// TIA Portal project "Serial_FB" (V15)

(* hardware
DEVICE "S7-1200 station_1"  S7-1200 Station
   slot 0: "Rack_0"  S7-1200 Rack  Rack  V1.0
   slot 1: "PLC_1"  CPU 1215C DC/DC/DC  6ES7 215-1AG40-0XB0  V4.2
DEVICE "HMI_1"  TP1200 Comfort
   slot 0: "HMI_1"  TP1200 Comfort  6AV2 124-0MC01-0AX0  15.0.0.0
   slot 1: "HMI_RT_1"  TP1200 Comfort  6AV2 124-0MC01-0AX0  15.0.0.0
   slot 5: "HMI_1.IE_CP_1"  PROFINET Interface  15.0.0.0
      slot 1: "PROFINET Interface_1"  PROFINET Interface
         slot 1: "Port_1"  Port
         slot 2: "Port_2"  Port
   slot 7: "HMI_1.MPI/DP_CP_1"  MPI/DP Interface  15.0.0.0
*)

// ===== PLC "PLC_1"  CPU 1215C DC/DC/DC =====

VAR_GLOBAL   // PLC tag table "Default tag table"
   "Begin_M" AT %M0.0 : Bool;
   "Pin_Out" AT %Q0.0 : Bool;
   "Port_Out" AT %QB0 : SInt;
   "Transfer_Status" AT %M0.1 : Bool;
   "Receive_Status" AT %M0.2 : Bool;
   "Start_M" AT %M0.3 : Bool;
   "Received_Byte" AT %MB2 : Byte;
END_VAR

DATA_BLOCK "Transmit_DB"   // DB2
{ S7_Optimized_Access := 'TRUE' }
VERSION : 0.1
// stored: InstanceOfName Transmit
"Transmit"
BEGIN
END_DATA_BLOCK

DATA_BLOCK "Receive_DB"   // DB4
{ S7_Optimized_Access := 'TRUE' }
VERSION : 0.1
// stored: InstanceOfName Receive
"Receive"
BEGIN
END_DATA_BLOCK

DATA_BLOCK "Input_48_Bit"   // DB5
{ S7_Optimized_Access := 'TRUE' }
VERSION : 0.1
   VAR RETAIN
      DI : Array[0..47] of Bool;
   END_VAR
BEGIN
END_DATA_BLOCK

// folder: System blocks/Program resources

DATA_BLOCK "Timer_1"   // DB1
{ S7_Optimized_Access := 'TRUE' }
AUTHOR : Simatic
FAMILY : IEC
NAME : IEC_TMR
VERSION : 1.0
// stored: InstanceOfName IEC_TIMER
"IEC_TIMER"
BEGIN
END_DATA_BLOCK

DATA_BLOCK "Timer_2"   // DB3
{ S7_Optimized_Access := 'TRUE' }
AUTHOR : Simatic
FAMILY : IEC
NAME : IEC_TMR
VERSION : 1.0
// stored: InstanceOfName IEC_TIMER
"IEC_TIMER"
BEGIN
END_DATA_BLOCK

// folder: (top level)

FUNCTION_BLOCK "Transmit"   // FB1, LAD
TITLE = Transmit 1 byte data serially to an output pin
{ S7_Optimized_Access := 'TRUE' }
VERSION : 0.1
   VAR_INPUT
      Data_In : Byte;
      "Begin" : Bool;
   END_VAR
   VAR_OUTPUT
      Serial_Out : Bool;
      Status : Bool;   // 1=In Progress, 0=Idle
   END_VAR
   VAR RETAIN
      Buffer : Array[0..9] of Bool;
      Temp : Byte;
      Clock : Time;
      i : DInt;
   END_VAR
   VAR_TEMP   // added for the SCL form of the ladder/FBD networks
      _w1 : Bool;
   END_VAR
   // Buffer[0] := true;
BEGIN

REGION Network 1: 1st bit of the input data
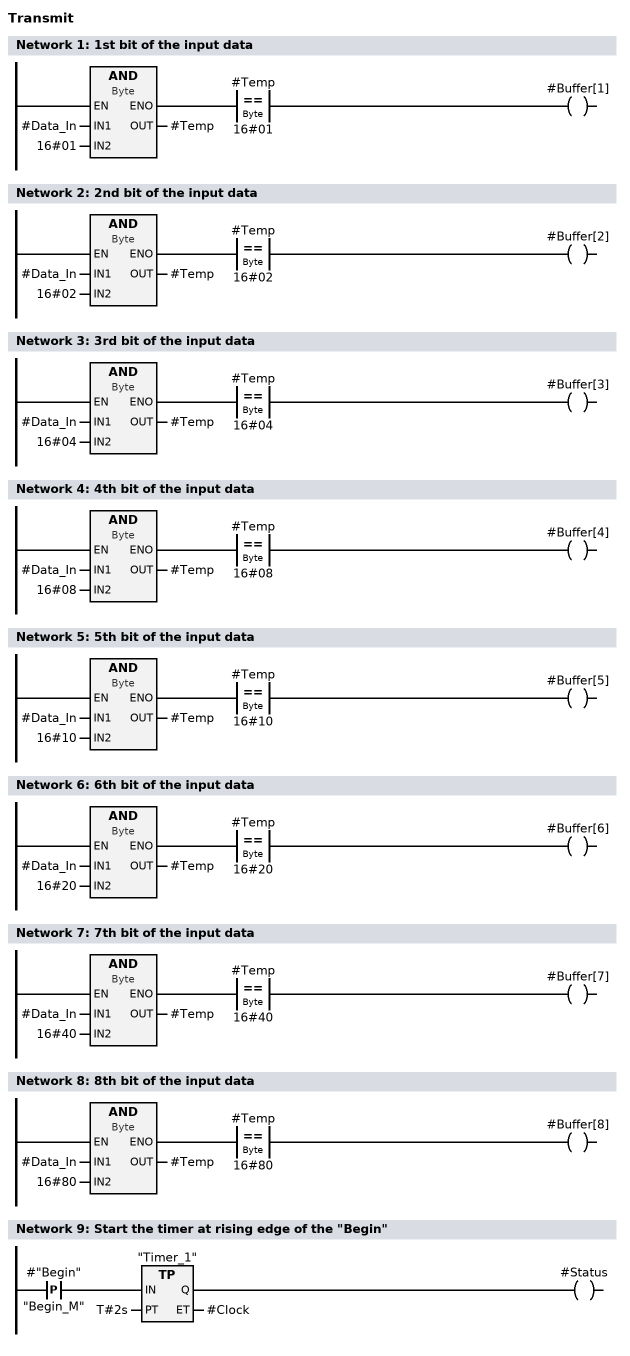
   RUNG wire#powerrail
      { S7_Templates := "SrcType := Byte" } And(in1 := #Data_In, in2 := 16#01, out => #Temp)
      { S7_Templates := "SrcType := Byte" } EQ_Contact(in1 := #Temp, in2 := 16#01)
      Coil( #Buffer[1] )
   END_RUNG
   // the same network as SCL:
   #Temp := #Data_In AND 16#01;
   #Buffer[1] := #Temp = 16#01;
END_REGION

REGION Network 2: 2nd bit of the input data
   RUNG wire#powerrail
      { S7_Templates := "SrcType := Byte" } And(in1 := #Data_In, in2 := 16#02, out => #Temp)
      { S7_Templates := "SrcType := Byte" } EQ_Contact(in1 := #Temp, in2 := 16#02)
      Coil( #Buffer[2] )
   END_RUNG
   // the same network as SCL:
   #Temp := #Data_In AND 16#02;
   #Buffer[2] := #Temp = 16#02;
END_REGION

REGION Network 3: 3rd bit of the input data
   RUNG wire#powerrail
      { S7_Templates := "SrcType := Byte" } And(in1 := #Data_In, in2 := 16#04, out => #Temp)
      { S7_Templates := "SrcType := Byte" } EQ_Contact(in1 := #Temp, in2 := 16#04)
      Coil( #Buffer[3] )
   END_RUNG
   // the same network as SCL:
   #Temp := #Data_In AND 16#04;
   #Buffer[3] := #Temp = 16#04;
END_REGION

REGION Network 4: 4th bit of the input data
   RUNG wire#powerrail
      { S7_Templates := "SrcType := Byte" } And(in1 := #Data_In, in2 := 16#08, out => #Temp)
      { S7_Templates := "SrcType := Byte" } EQ_Contact(in1 := #Temp, in2 := 16#08)
      Coil( #Buffer[4] )
   END_RUNG
   // the same network as SCL:
   #Temp := #Data_In AND 16#08;
   #Buffer[4] := #Temp = 16#08;
END_REGION

REGION Network 5: 5th bit of the input data
   RUNG wire#powerrail
      { S7_Templates := "SrcType := Byte" } And(in1 := #Data_In, in2 := 16#10, out => #Temp)
      { S7_Templates := "SrcType := Byte" } EQ_Contact(in1 := #Temp, in2 := 16#10)
      Coil( #Buffer[5] )
   END_RUNG
   // the same network as SCL:
   #Temp := #Data_In AND 16#10;
   #Buffer[5] := #Temp = 16#10;
END_REGION

REGION Network 6: 6th bit of the input data
   RUNG wire#powerrail
      { S7_Templates := "SrcType := Byte" } And(in1 := #Data_In, in2 := 16#20, out => #Temp)
      { S7_Templates := "SrcType := Byte" } EQ_Contact(in1 := #Temp, in2 := 16#20)
      Coil( #Buffer[6] )
   END_RUNG
   // the same network as SCL:
   #Temp := #Data_In AND 16#20;
   #Buffer[6] := #Temp = 16#20;
END_REGION

REGION Network 7: 7th bit of the input data
   RUNG wire#powerrail
      { S7_Templates := "SrcType := Byte" } And(in1 := #Data_In, in2 := 16#40, out => #Temp)
      { S7_Templates := "SrcType := Byte" } EQ_Contact(in1 := #Temp, in2 := 16#40)
      Coil( #Buffer[7] )
   END_RUNG
   // the same network as SCL:
   #Temp := #Data_In AND 16#40;
   #Buffer[7] := #Temp = 16#40;
END_REGION

REGION Network 8: 8th bit of the input data
   RUNG wire#powerrail
      { S7_Templates := "SrcType := Byte" } And(in1 := #Data_In, in2 := 16#80, out => #Temp)
      { S7_Templates := "SrcType := Byte" } EQ_Contact(in1 := #Temp, in2 := 16#80)
      Coil( #Buffer[8] )
   END_RUNG
   // the same network as SCL:
   #Temp := #Data_In AND 16#80;
   #Buffer[8] := #Temp = 16#80;
END_REGION

REGION Network 9: Start the timer at rising edge of the "Begin"
   #_w1 := #"Begin" AND NOT "Begin_M";   // rising edge of #"Begin"
   "Begin_M" := #"Begin";
   "Timer_1".TP(IN := #_w1, PT := T#2s, ET => #Clock);
   #Status := "Timer_1".Q;
END_REGION

REGION Network 10 (SCL): Transmission of "Buffer"
   IF #Status THEN

       #i := TIME_TO_DINT(#Clock)/200;
       #Serial_Out := #Buffer[#i];

   //    IF #Clock > T#0ms AND #Clock < T#200ms THEN
   //        #Serial_Out := #Buffer[0];
   //    END_IF;

   END_IF;
END_REGION
END_FUNCTION_BLOCK

FUNCTION_BLOCK "Receive"   // FB2, LAD
TITLE = Serial Receiver Block
{ S7_Optimized_Access := 'TRUE' }
VERSION : 0.1
   VAR_INPUT
      Serial_In : Bool;
   END_VAR
   VAR_OUTPUT
      Data_Out : Byte;
      Status : Bool;   // 1=In Progress, 0=Idle
   END_VAR
   VAR RETAIN
      Buffer : Array[0..9] of Bool;
      Temp : Byte;
      Clock : Time;
      i : DInt;
      j : Byte;
      k : SInt;
   END_VAR
   VAR_TEMP   // added for the SCL form of the ladder/FBD networks
      _w1 : Bool;
   END_VAR
BEGIN

REGION Network 1: Start timer for data reception
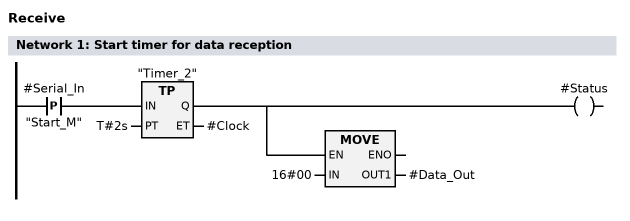
   #_w1 := #Serial_In AND NOT "Start_M";   // rising edge of #Serial_In
   "Start_M" := #Serial_In;
   "Timer_2".TP(IN := #_w1, PT := T#2s, ET => #Clock);
   #Status := "Timer_2".Q;
   IF "Timer_2".Q THEN #Data_Out := 16#00; END_IF;
END_REGION

REGION Network 2 (SCL): Data reception and storage in buffer
   IF #Status THEN

       #i := TIME_TO_DINT(#Clock) / 200;
       IF TIME_TO_DINT(#Clock) = (#i*200)+100 THEN
           #Buffer[#i] := #Serial_In;
       END_IF;

       //    IF #Clock > T#0ms AND #Clock < T#200ms THEN
       //        #Serial_Out := #Buffer[0];
       //    END_IF;

   END_IF;
END_REGION

REGION Network 3 (SCL): Data storage in the variable "Data_Out"
   FOR #k := 1 TO 8 DO
       #j := BOOL_TO_BYTE(#Buffer[#k]);
       #j := SHL(IN := #j, N := (SINT_TO_USINT(#k - 1)));
       #Data_Out := #Data_Out OR #j;
   END_FOR;
END_REGION
END_FUNCTION_BLOCK

ORGANIZATION_BLOCK "Main"   // OB1, LAD, ProgramCycle
TITLE = "Main Program Sweep (Cycle)"
{ S7_Optimized_Access := 'TRUE' }
VERSION : 0.1
   VAR_INPUT
      Initial_Call : Bool;   // Initial call of this OB
      Remanence : Bool;   // =True, if remanent data are available
   END_VAR
BEGIN

REGION Network 1
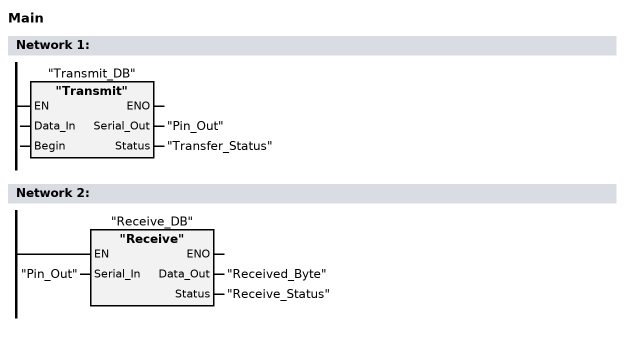
   RUNG wire#powerrail
      "Transmit_DB"(Data_In :=, "Begin" :=, Serial_Out => "Pin_Out", Status => "Transfer_Status")
   END_RUNG
   // the same network as SCL:
   "Transmit_DB"(Serial_Out => "Pin_Out", Status => "Transfer_Status");   // "Transmit"
END_REGION

REGION Network 2
   RUNG wire#powerrail
      "Receive_DB"(Serial_In := "Pin_Out", Data_Out => "Received_Byte", Status => "Receive_Status")
   END_RUNG
   // the same network as SCL:
   "Receive_DB"(Serial_In := "Pin_Out", Data_Out => "Received_Byte", Status => "Receive_Status");   // "Receive"
END_REGION
END_ORGANIZATION_BLOCK

(* ===== HMI "HMI_RT_1" =====
system functions are stored by id; their names below are inferred from use
connection "HMI_Connection_1": ETHERNET, S7_1200_OMS

HMI tags "Default tag table"
   "Tag_ScreenNumber" : UInt, internal
   "Port_Out" : SInt = PLC Port_Out AT %QB0, 100 ms

screen "Root screen" 1280x740, template "Template_1"
   on GenerateScreen: SetTag("Tag_ScreenNumber", 1)
   TrendView "Trend view_1" at 3,2 size 1275x676

Template "Template_1" 1280x740
   Button "Exit" at 1200,679 size 78x59; TextOff 'Exit'; PictureOff "ExitRuntime_TP1200_Comfort_TR"; PictureOn "ExitRuntime_TP1200_Comfort_TR"
      on Release: StopRuntime(0)
   Button "Template_Button" at 1120,679 size 78x59; TextOff 'Text'
   Button "Template_Button_1" at 1040,679 size 78x59; TextOff 'Text'
   Button "Template_Button_2" at 960,679 size 78x59; TextOff 'Text'
   Button "Template_Button_3" at 880,679 size 78x59; TextOff 'Text'
   Button "Template_Button_4" at 800,679 size 78x59; TextOff 'Text'
   Button "Template_Button_5" at 720,679 size 78x59; TextOff 'Text'
   Button "Template_Button_6" at 640,679 size 78x59; TextOff 'Text'
   Button "Template_Button_7" at 561,679 size 78x59; TextOff 'Text'
   Button "Template_Button_8" at 481,679 size 78x59; TextOff 'Text'
   Button "Template_Button_9" at 401,679 size 78x59; TextOff 'Text'
   Button "Template_Button_10" at 321,679 size 78x59; TextOff 'Text'
   Button "Template_Button_11" at 241,679 size 78x59; TextOff 'Text'
   Button "Template_Button_12" at 161,679 size 78x59; TextOff 'Text'
   Button "Alarms" at 81,679 size 78x59; TextOff 'Alarms'; PictureOff "AlarmDisplay_TP1200_Comfort_TR"; PictureOn "AlarmDisplay_TP1200_Comfort_TR"
      on Release: function_ef3f5d25("Alarm window_Unacknowledged", -1)
   Button "Start screen" at 1,679 size 78x59; TextOff 'Start screen'; PictureOff "NavigateHome_TP1200_Comfort_TR"; PictureOn "NavigateHome_TP1200_Comfort_TR"
      on Release: ActivateScreen("Root screen", 0)
*)